PROGRAM MAIN
VAR
	bEnable : BOOL;
	bStart : BOOL;
	nInt : INT := -32768;
	nUint : UINT := 65535;
	fReal : REAL := 255.255;
	sPowerstatus : STRING := 'Power Off';
	
    nFloatConversion : INT;
	fFloatConversion : LREAL;
	nHeltall : INT:= 100;
	fKomma : LREAL := 100.5;
	
END_VAR

bEnable := bStart;

nFloatConversion := nHeltall + LREAL_TO_INT(fKomma);

END_PROGRAM

(* stored: Version 1.1.0.1, ProductVersion 3.1.4024.12
   POU MAIN: Id {a0431b7a-35bf-4913-a95a-838fe599a7d8}, SpecialFunc None *)
